// TwinCAT 3 PLC project test
// ProgramVersion: 3.1.4020.5
// libraries:
//   L2Si Vacuum Library, * (SLAC)
//   LCLS General, * (SLAC)
//   Tc2_Standard, * (Beckhoff Automation GmbH)
//   Tc2_System, * (Beckhoff Automation GmbH)
//   Tc3_Module, * (Beckhoff Automation GmbH)
//   PMPS,newest,SLAC - LCLS
// project tree:
//   GVLs/ GVL_Devices.TcGVL, GVL_PMPS.TcGVL
//   / PlcTask.TcTTO
//   POUs/ MAIN.TcPOU
// real-time tasks:
//   TASK PlcTask: cycle T#10ms, priority 20, ADS port 350
// I/O:
//   DEVICE Device 1 (EtherCAT) (disabled), AmsNetId 172.21.148.215.2.1
//     Term 1 (EK1100) [EK1100 EtherCAT Coupler (2A E-Bus)]
//       Term 2 (EL3174-0002) [EL3174-0002 4Ch. Ana. Input +/-10V, +/-20mA 16 Bit, Isolated Channels]
//       Term 3 (EL3174-0002) [EL3174-0002 4Ch. Ana. Input +/-10V, +/-20mA 16 Bit, Isolated Channels]
//       Term 4 (EL2624) [EL2624 4Ch. Relay Output, NO (125V AC / 30V DC)]
//       Term 6 (EL1004) [EL1004 4Ch. Dig. Input 24V, 3ms]
//       Term 5 (EL1004) [EL1004 4Ch. Dig. Input 24V, 3ms]
//       Term 7 (EL2004) [EL2004 4Ch. Dig. Output 24V, 0.5A]
//       Term 8 (EL3064) [EL3064 4Ch. Ana. Input 0-10V]
//       Term 9 (EL2794) [EL2794 4Ch. Dig. Output 24V AC/DC, 2A, short-circuit-proof]
//       Term 10 (EL1004) [EL1004 4Ch. Dig. Input 24V, 3ms]
//       Term 11 (EL1124) [EL1124 4Ch. Dig. Input 5V, 10µs, Sensor Power]
//       Term 12 (EL1124) [EL1124 4Ch. Dig. Input 5V, 10µs, Sensor Power]
//       Term 13 (EL3064) [EL3064 4Ch. Ana. Input 0-10V]

CONFIGURATION test
    RESOURCE PLC ON TwinCAT3
        TASK PlcTask(INTERVAL := T#10ms, PRIORITY := 20);
        PROGRAM MAIN WITH PlcTask : MAIN;
    END_RESOURCE
END_CONFIGURATION

// ---- GVLs/GVL_Devices.TcGVL
VAR_GLOBAL
	{attribute 'pytmc' := '
    pv: FEE:VGC:02
	'}
	FEE_VGC_02: FB_VGC;
	{attribute 'pytmc' := '
    pv: FEE:KMONO:GPI:01
	'}
	FEE_KMONO_GPI_01: FB_MKS275;
	{attribute 'pytmc' := '
    pv: FEE:KMONO:GCC:01
	'}
	FEE_KMONO_GCC_01: FB_MKS500;
	{attribute 'pytmc' := '
    pv: FEE:KMONO:PIP:01
	'}
	FEE_KMONO_PIP_01: FB_PIP_Gamma;
	{attribute 'pytmc' := '
    pv: FEE:PIP:02
	'}
	FEE_PIP_02: FB_PIP_Gamma;
	{attribute 'pytmc' := '
    pv: FEE:GPI:03
	'}
	FEE_GPI_03: FB_MKS275;
	{attribute 'pytmc' := '
    pv: FEE:GCC:03
	'}
	FEE_GCC_03: FB_MKS500;
	{attribute 'pytmc' := '
    pv: FEE:VGC:03
	'}
	FEE_VGC_03: FB_VGC;
	{attribute 'pytmc' := '
    pv: FEE:M1L:GPI:01
	'}
	FEE_M1L_GPI_01: FB_MKS275;
	{attribute 'pytmc' := '
    pv: FEE:M1L:GCC:03
	'}
	FEE_M1L_GCC_01: FB_MKS500;
	{attribute 'pytmc' := '
    pv: FEE:M1L:PIP:01
	'}
	FEE_M1L_PIP_01: FB_PIP_Gamma;
	{attribute 'pytmc' := '
    pv: FEE:PIP:03
	'}
	FEE_PIP_03: FB_PIP_Gamma;
	{attribute 'pytmc' := '
    pv: FEE:GPI:04
	'}
	FEE_GPI_04: FB_MKS275;
	{attribute 'pytmc' := '
    pv: FEE:GCC:04
	'}
	FEE_GCC_04: FB_MKS500;
	{attribute 'pytmc' := '
    pv: FEE:VGC:04
	'}
	FEE_VGC_04: FB_VGC;
	
END_VAR

// ---- GVLs/GVL_PMPS.TcGVL

VAR_GLOBAL
	
{attribute 'pytmc' := '
    pv: PLC:TST:FF1
    '}
    {attribute 'TcLinkTo' := '.q_xFastFaultOut:=TIIB[PMPS_FFO]^Channel 1^Output'}
    g_FastFaultOutput1  :   FB_HardwareFFOutput;
	
	{attribute 'pytmc' := '
    pv: PLC:TST:FF2
    '}
    {attribute 'TcLinkTo' := '.q_xFastFaultOut:=TIIB[PMPS_FFO]^Channel 2^Output'}
    g_FastFaultOutput2  :   FB_HardwareFFOutput;
END_VAR

// ---- POUs/MAIN.TcPOU
PROGRAM MAIN
VAR

END_VAR


//valves
FEE_VGC_02(
	i_stUSG:= FEE_KMONO_GCC_01.IG, 
	i_stDSG:= FEE_KMONO_GCC_01.IG , 
	i_xDis_DPIlk:= FALSE, 
	i_xEPS_OK:= FALSE, 
	i_xPMPS_OK:= , 
	i_xExt_OK:= TRUE, 
	i_xOverrideMode:= , 
	i_xReset:= , 
	iq_stValve=> , 
	xMPS_OK=> , 
	io_fbFFHWO:= g_FastFaultOutput1 );

FEE_VGC_03(
	i_stUSG:=FEE_KMONO_GCC_01.IG, 
	i_stDSG:= FEE_M1L_GCC_01.IG , 
	i_xDis_DPIlk:= FALSE, 
	i_xEPS_OK:= FALSE, 
	i_xPMPS_OK:= TRUE, 
	i_xExt_OK:= TRUE, 
	i_xOverrideMode:= , 
	i_xReset:= , 
	iq_stValve=> , 
	xMPS_OK=> , 
	io_fbFFHWO:= g_FastFaultOutput1 );

FEE_VGC_04(
	i_stUSG:= FEE_GCC_03.IG, 
	i_stDSG:= FEE_GCC_03.IG , 
	i_xDis_DPIlk:= FALSE, 
	i_xEPS_OK:= FALSE, 
	i_xPMPS_OK:= TRUE, 
	i_xExt_OK:= TRUE, 
	i_xOverrideMode:= , 
	i_xReset:= , 
	iq_stValve=> , 
	xMPS_OK=> , 
	io_fbFFHWO:= g_FastFaultOutput1 );	
	
// gauges and pip
FEE_KMONO_GPI_01(PG=>);
FEE_KMONO_GCC_01(PG:=FEE_KMONO_GPI_01.PG);
FEE_KMONO_PIP_01(i_stGauge:= FEE_KMONO_GCC_01.IG);

FEE_GPI_03(PG=>);
FEE_GCC_03(PG:=FEE_KMONO_GPI_01.PG);

FEE_PIP_02(i_stGauge:= FEE_GCC_03.IG);

FEE_M1L_GPI_01(PG=>);
FEE_M1L_GCC_01(PG:=FEE_M1L_GPI_01.PG);
FEE_M1L_PIP_01(i_stGauge:= FEE_M1L_GCC_01.IG);

FEE_GPI_04(PG=>);
FEE_GCC_04(PG:=FEE_GPI_04.PG);
FEE_PIP_03(i_stGauge:= FEE_GCC_04.IG);

END_PROGRAM
